FUNCTION BufferRealToReal : REAL
VAR_INPUT
	raw_input : REAL;
END_VAR
VAR_OUTPUT
	real_output : REAL;
END_VAR
VAR
	temp: REAL;
END_VAR

temp := raw_input;
MEMCPY(ADR(real_output), ADR(temp), SIZEOF(temp));

END_FUNCTION

(* stored: Version 1.1.0.1, ProductVersion 3.1.4024.9
   POU BufferRealToReal: Id {c8b73249-0fa5-4065-8cbc-01e649bbb727}, SpecialFunc None *)
